PROGRAM NET_VAR_MASTER_DEMO
VAR
	NET_VAR_CONTROL_1: NET_VAR_CONTROL;
	activate: BOOL := TRUE;
	run: BOOL;
	udp: BOOL := TRUE;
	master: BOOL := TRUE;
	remote_port: WORD := 10000;
	scan_time: TIME := T#1s;
	watchdog: TIME := T#2s;
	error: DWORD;
	x: NET_VAR_DATA;

	NET_VAR_BOOL8_1: NET_VAR_BOOL8;
	id_b8: BYTE;
	in_b1: BOOL;
	in_b2: BOOL;
	in_b3: BOOL;
	in_b4: BOOL;
	in_b5: BOOL;
	in_b6: BOOL;
	in_b7: BOOL;
	in_b8: BOOL;
	out_b1: BOOL;
	out_b2: BOOL;
	out_b3: BOOL;
	out_b4: BOOL;
	out_b5: BOOL;
	out_b6: BOOL;
	out_b7: BOOL;
	out_b8: BOOL;

	NET_VAR_STRING_1: NET_VAR_STRING;
	in_s1: T_MaxString;
	out_s1: T_MaxString;
	id_s: BYTE;

	NET_VAR_BUFFER_1: NET_VAR_BUFFER;
	id_bu: BYTE;
	BUF_IN : ARRAY [1..64] OF BYTE;
	BUF_OUT : ARRAY [1..64] OF BYTE;

	id_dw: BYTE;
	NET_VAR_DWORD8_1: NET_VAR_DWORD8;
	in_dw1 : DWORD;
	in_dw2 : DWORD;
	in_dw3 : DWORD;
	in_dw4 : DWORD;
	in_dw5 : DWORD;
	in_dw6 : DWORD;
	in_dw7 : DWORD;
	in_dw8 : DWORD;
	out_dw1 : DWORD;
	out_dw2 : DWORD;
	out_dw3 : DWORD;
	out_dw4 : DWORD;
	out_dw5 : DWORD;
	out_dw6 : DWORD;
	out_dw7 : DWORD;
	out_dw8 : DWORD;

	NET_VAR_REAL8_1: NET_VAR_REAL8;
	in_r1 : REAL;
	in_r2 : REAL;
	in_r3 : REAL;
	in_r4 : REAL;
	in_r5 : REAL;
	in_r6 : REAL;
	in_r7 : REAL;
	in_r8 : REAL;
	out_r1 : REAL;
	out_r2 : REAL;
	out_r3 : REAL;
	out_r4 : REAL;
	out_r5 : REAL;
	out_r6 : REAL;
	out_r7 : REAL;
	out_r8 : REAL;
	id_r: BYTE;

	NET_VAR_X8_1: NET_VAR_X8;
	in_x_re1 : REAL;
	in_x_re2 : REAL;
	in_x_di1 : DINT;
	in_x_di2 : DINT;
	in_x_ud1 : UDINT;
	in_x_ud2 : UDINT;
	in_x_dw1 : DWORD;
	in_x_dw2 : DWORD;
	out_x_re1 : REAL;
	out_x_re2 : REAL;
	out_x_di1 : DINT;
	out_x_di2 : DINT;
	out_x_ud1 : UDINT;
	out_x_ud2 : UDINT;
	out_x_dw1 : DWORD;
	out_x_dw2 : DWORD;
	id_x8: BYTE;
END_VAR
VAR // added by the converter: edge detectors and wires of the graphical bodies
    _w1 : ANY;
END_VAR

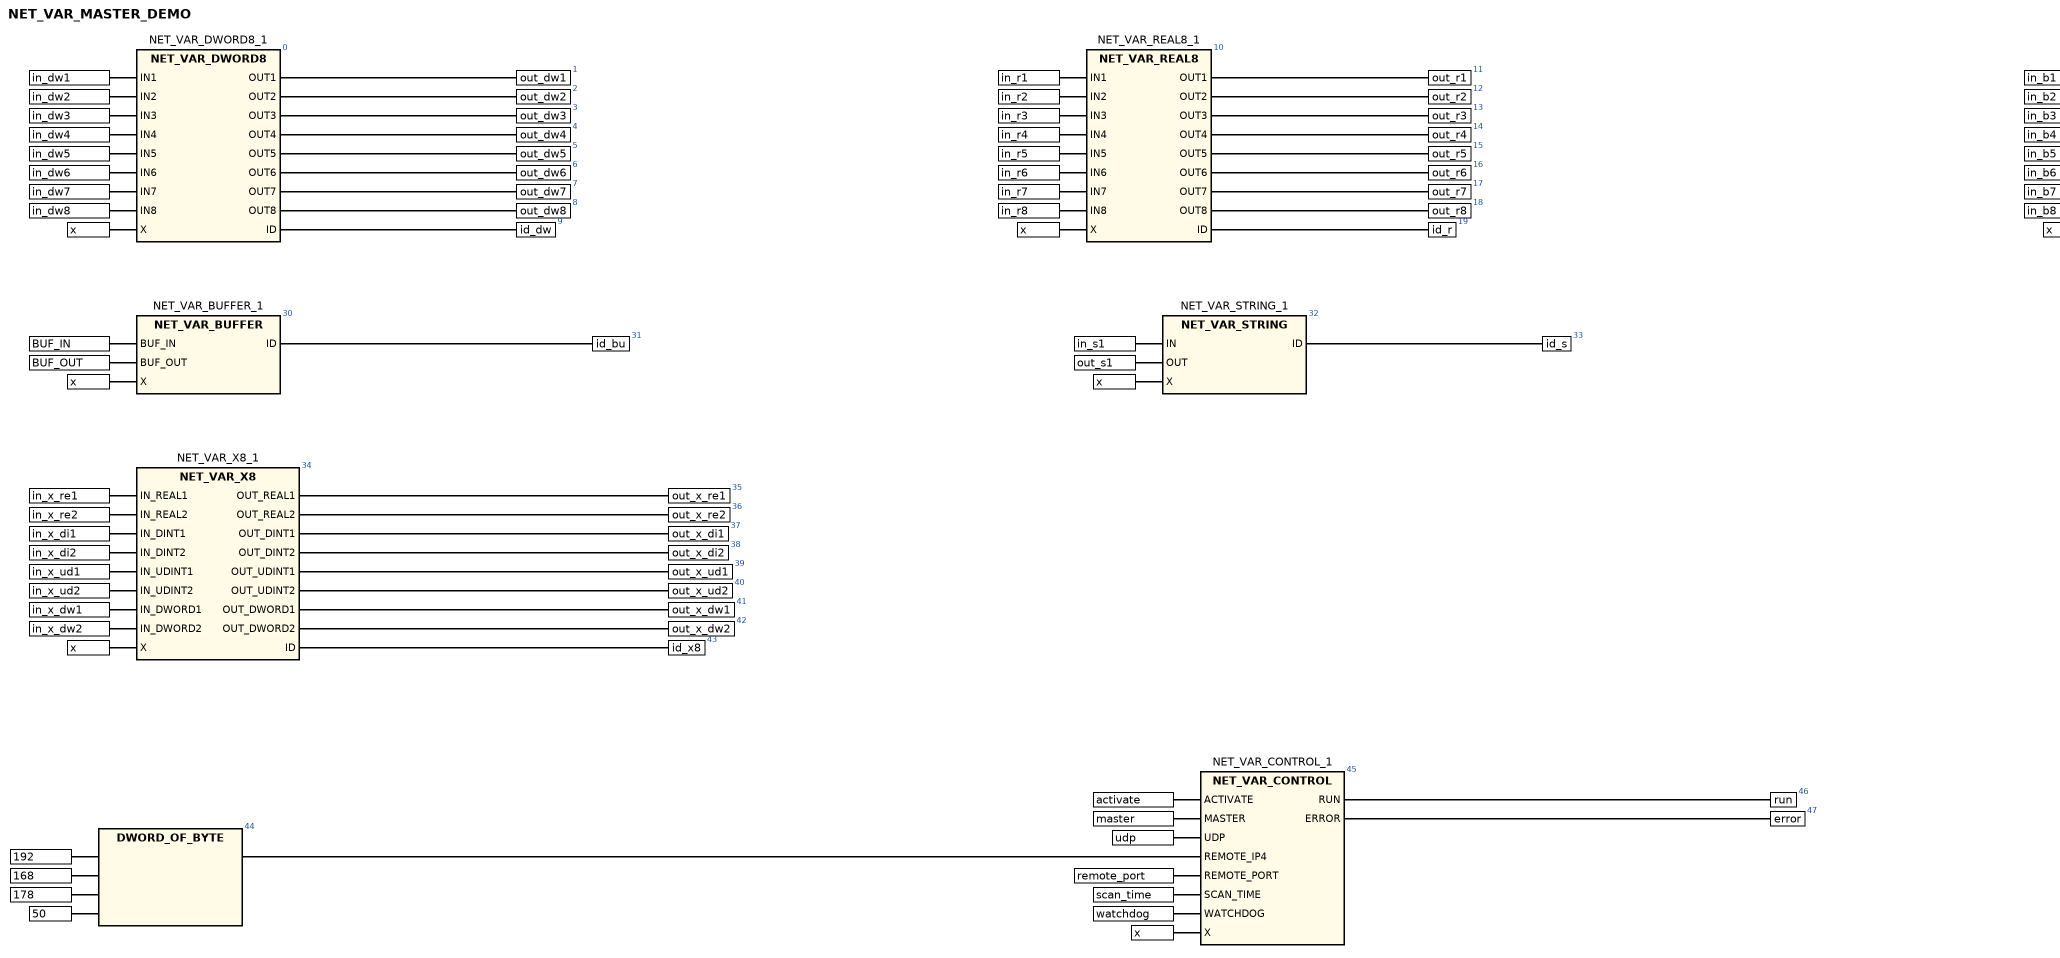
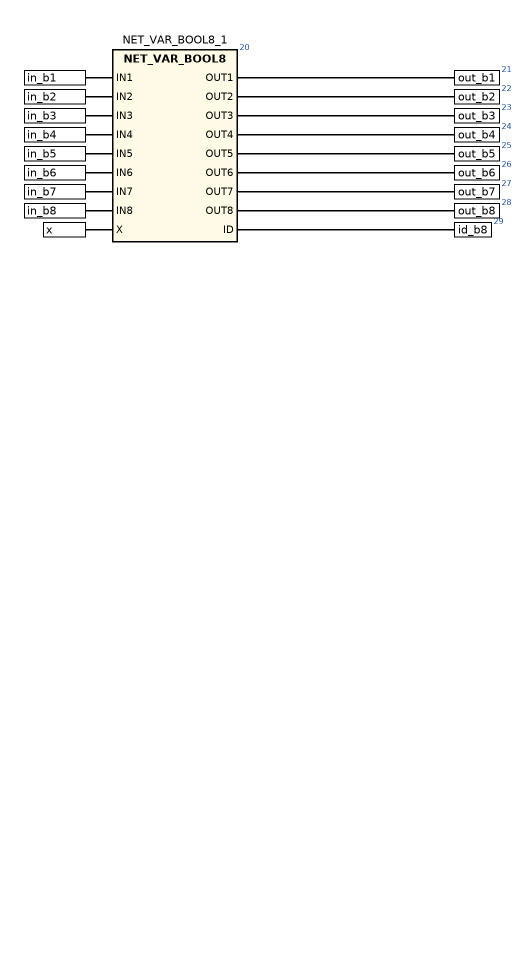
NET_VAR_DWORD8_1(
    IN1 := in_dw1,
    IN2 := in_dw2,
    IN3 := in_dw3,
    IN4 := in_dw4,
    IN5 := in_dw5,
    IN6 := in_dw6,
    IN7 := in_dw7,
    IN8 := in_dw8,
    X := x); // NET_VAR_DWORD8
out_dw1 := NET_VAR_DWORD8_1.OUT1;
out_dw2 := NET_VAR_DWORD8_1.OUT2;
out_dw3 := NET_VAR_DWORD8_1.OUT3;
out_dw4 := NET_VAR_DWORD8_1.OUT4;
out_dw5 := NET_VAR_DWORD8_1.OUT5;
out_dw6 := NET_VAR_DWORD8_1.OUT6;
out_dw7 := NET_VAR_DWORD8_1.OUT7;
out_dw8 := NET_VAR_DWORD8_1.OUT8;
id_dw := NET_VAR_DWORD8_1.ID;
NET_VAR_REAL8_1(
    IN1 := in_r1,
    IN2 := in_r2,
    IN3 := in_r3,
    IN4 := in_r4,
    IN5 := in_r5,
    IN6 := in_r6,
    IN7 := in_r7,
    IN8 := in_r8,
    X := x); // NET_VAR_REAL8
out_r1 := NET_VAR_REAL8_1.OUT1;
out_r2 := NET_VAR_REAL8_1.OUT2;
out_r3 := NET_VAR_REAL8_1.OUT3;
out_r4 := NET_VAR_REAL8_1.OUT4;
out_r5 := NET_VAR_REAL8_1.OUT5;
out_r6 := NET_VAR_REAL8_1.OUT6;
out_r7 := NET_VAR_REAL8_1.OUT7;
out_r8 := NET_VAR_REAL8_1.OUT8;
id_r := NET_VAR_REAL8_1.ID;
NET_VAR_BOOL8_1(
    IN1 := in_b1,
    IN2 := in_b2,
    IN3 := in_b3,
    IN4 := in_b4,
    IN5 := in_b5,
    IN6 := in_b6,
    IN7 := in_b7,
    IN8 := in_b8,
    X := x); // NET_VAR_BOOL8
out_b1 := NET_VAR_BOOL8_1.OUT1;
out_b2 := NET_VAR_BOOL8_1.OUT2;
out_b3 := NET_VAR_BOOL8_1.OUT3;
out_b4 := NET_VAR_BOOL8_1.OUT4;
out_b5 := NET_VAR_BOOL8_1.OUT5;
out_b6 := NET_VAR_BOOL8_1.OUT6;
out_b7 := NET_VAR_BOOL8_1.OUT7;
out_b8 := NET_VAR_BOOL8_1.OUT8;
id_b8 := NET_VAR_BOOL8_1.ID;
NET_VAR_BUFFER_1(BUF_IN := BUF_IN, BUF_OUT := BUF_OUT, X := x); // NET_VAR_BUFFER
id_bu := NET_VAR_BUFFER_1.ID;
NET_VAR_STRING_1(IN := in_s1, OUT := out_s1, X := x); // NET_VAR_STRING
id_s := NET_VAR_STRING_1.ID;
NET_VAR_X8_1(
    IN_REAL1 := in_x_re1,
    IN_REAL2 := in_x_re2,
    IN_DINT1 := in_x_di1,
    IN_DINT2 := in_x_di2,
    IN_UDINT1 := in_x_ud1,
    IN_UDINT2 := in_x_ud2,
    IN_DWORD1 := in_x_dw1,
    IN_DWORD2 := in_x_dw2,
    X := x); // NET_VAR_X8
out_x_re1 := NET_VAR_X8_1.OUT_REAL1;
out_x_re2 := NET_VAR_X8_1.OUT_REAL2;
out_x_di1 := NET_VAR_X8_1.OUT_DINT1;
out_x_di2 := NET_VAR_X8_1.OUT_DINT2;
out_x_ud1 := NET_VAR_X8_1.OUT_UDINT1;
out_x_ud2 := NET_VAR_X8_1.OUT_UDINT2;
out_x_dw1 := NET_VAR_X8_1.OUT_DWORD1;
out_x_dw2 := NET_VAR_X8_1.OUT_DWORD2;
id_x8 := NET_VAR_X8_1.ID;
_w1 := DWORD_OF_BYTE(192, 168, 178, 50);
NET_VAR_CONTROL_1(
    ACTIVATE := activate,
    MASTER := master,
    UDP := udp,
    REMOTE_IP4 := _w1,
    REMOTE_PORT := remote_port,
    SCAN_TIME := scan_time,
    WATCHDOG := watchdog,
    X := x); // NET_VAR_CONTROL
run := NET_VAR_CONTROL_1.RUN;
error := NET_VAR_CONTROL_1.ERROR;

END_PROGRAM

(* stored: Version 1.1.0.1, ProductVersion 3.1.4024.9
   POU NET_VAR_MASTER_DEMO: Id {1a39ad8b-5591-48d2-84b3-16aa070c705e}, SpecialFunc None *)
